% RSLogix 500 project ACNASR.RSS, saved by version 9.00.00.04 %
PROJECT "UNTITLED"    % processor: Bul.1763 MicroLogix 1100 Series B %

PROGRAM FILES
  LAD 2   5 rungs

DATA FILES
  O0 OUTPUT  4 elements
  I1 INPUT  6 elements
  S2 STATUS  66 elements
  B3 BINARY  1 elements
  T4 TIMER  1 elements
  C5 COUNTER  1 elements
  R6 CONTROL  1 elements
  N7 INTEGER  3 elements
  F8 FLOAT  1 elements
  ST9 STRINGS  4 elements

LADDER 2
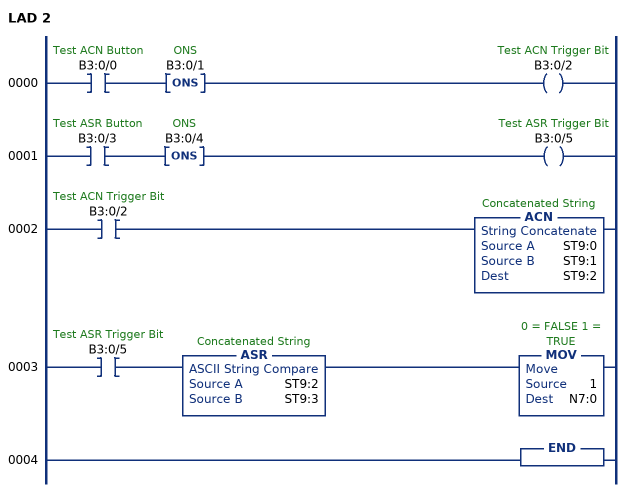
% Rung: 0 %
SOR XIC B3:0/0 ONS B3:0/1 OTE B3:0/2 EOR
%   B3:0/0  "Test ACN Button" %
%   B3:0/1  "ONS" %
%   B3:0/2  "Test ACN Trigger Bit" %
% Rung: 1 %
SOR XIC B3:0/3 ONS B3:0/4 OTE B3:0/5 EOR
%   B3:0/3  "Test ASR Button" %
%   B3:0/4  "ONS" %
%   B3:0/5  "Test ASR Trigger Bit" %
% Rung: 2 %
SOR XIC B3:0/2 ACN ST9:0 ST9:1 ST9:2 EOR
%   B3:0/2  "Test ACN Trigger Bit" %
%   ST9:0  "Partial String 1" %
%   ST9:1  "Partial String 2" %
%   ST9:2  "Concatenated String" %
% Rung: 3 %
SOR XIC B3:0/5 ASR ST9:2 ST9:3 MOV 1 N7:0 EOR
%   B3:0/5  "Test ASR Trigger Bit" %
%   ST9:2  "Concatenated String" %
%   ST9:3  "Test Value" %
%   N7:0  "0 = FALSE 1 = TRUE" %
% Rung: 4 %
SOR END EOR

DATA TABLE (non-zero values as saved)
DATA ST9
% ST9:0 % "TEST"
% ST9:1 % "STRING"
% ST9:2 % "SOMETHING"
% ST9:3 % "TESTSTRING"
